(* IEC 61131-3 sources: PLC_FB_Sequencer/, 4 files *)

(* ---- MachineState1.st ---- *)
(* ======================================== *)
(* State Machine:  *)
(* Author: 1.0 *)
(* Version:  *)
(* Generated: 2025-11-28 15:15:25 *)
(* ======================================== *)

FUNCTION_BLOCK

VAR_INPUT
    IN_01 : BOOL;
    IN_02 : BOOL;
    IN_03 : BOOL;
    IN_04 : BOOL;
    IN_05 : BOOL;
    IN_06 : BOOL;
    IN_07 : BOOL;
    IN_08 : BOOL;
    IN_09 : BOOL;
    IN_10 : BOOL;
    IN_11 : BOOL;
    IN_12 : BOOL;
    IN_13 : BOOL;
    IN_14 : BOOL;
    IN_15 : BOOL;
    IN_16 : BOOL;
END_VAR

VAR_OUTPUT
    OUT_01 : BOOL;
    OUT_02 : BOOL;
    OUT_03 : BOOL;
    OUT_04 : BOOL;
    OUT_05 : BOOL;
    OUT_06 : BOOL;
    OUT_07 : BOOL;
    OUT_08 : BOOL;
    OUT_09 : BOOL;
    OUT_10 : BOOL;
    OUT_11 : BOOL;
    OUT_12 : BOOL;
    OUT_13 : BOOL;
    OUT_14 : BOOL;
    OUT_15 : BOOL;
    OUT_16 : BOOL;
END_VAR

VAR
    currentState : (IDLE, STATE_2, STATE_3) := IDLE;
END_VAR

(* State Machine Logic *)
CASE currentState OF

    IDLE:
        (* Actions *)
        OUT_01 := FALSE;
        OUT_02 := FALSE;
        OUT_03 := FALSE;
        OUT_04 := FALSE;
        OUT_05 := FALSE;
        OUT_06 := FALSE;
        OUT_07 := FALSE;
        OUT_08 := FALSE;
        OUT_09 := FALSE;
        OUT_10 := FALSE;
        OUT_11 := FALSE;
        OUT_12 := FALSE;
        OUT_13 := FALSE;
        OUT_14 := FALSE;
        OUT_15 := FALSE;
        OUT_16 := FALSE;
        (* No actions *)

        (* Transitions *)
        IF IN_01 AND IN_02 THEN  (* Example transition *)
            currentState := STATE_2;
        END_IF;

    STATE_2:
        (* Actions *)
        OUT_01 := TRUE;
        OUT_02 := FALSE;
        OUT_03 := FALSE;
        OUT_04 := FALSE;
        OUT_05 := FALSE;
        OUT_06 := FALSE;
        OUT_07 := FALSE;
        OUT_08 := FALSE;
        OUT_09 := FALSE;
        OUT_10 := FALSE;
        OUT_11 := FALSE;
        OUT_12 := FALSE;
        OUT_13 := FALSE;
        OUT_14 := FALSE;
        OUT_15 := FALSE;
        OUT_16 := FALSE;
        (* No actions *)

        (* Transitions *)
        IF IN_03 THEN
            currentState := STATE_3;
        END_IF;

    STATE_3:
        (* Actions *)
        OUT_01 := TRUE;
        OUT_02 := TRUE;
        OUT_03 := FALSE;
        OUT_04 := FALSE;
        OUT_05 := FALSE;
        OUT_06 := FALSE;
        OUT_07 := FALSE;
        OUT_08 := FALSE;
        OUT_09 := FALSE;
        OUT_10 := FALSE;
        OUT_11 := FALSE;
        OUT_12 := FALSE;
        OUT_13 := FALSE;
        OUT_14 := FALSE;
        OUT_15 := FALSE;
        OUT_16 := FALSE;
        (* No actions *)

        (* Transitions *)
        IF NOT IN_01 THEN
            currentState := IDLE;
        END_IF;
END_CASE;

END_FUNCTION_BLOCK

(* ---- MachineState2.st ---- *)
(* ======================================== *)
(* State Machine:  *)
(* Author: 1.0 *)
(* Version:  *)
(* Generated: 2025-11-29 16:41:58 *)
(* ======================================== *)

FUNCTION_BLOCK

VAR_INPUT
    IN_01 : BOOL;
    IN_02 : BOOL;
    IN_03 : BOOL;
    IN_04 : BOOL;
    IN_05 : BOOL;
    IN_06 : BOOL;
    IN_07 : BOOL;
    IN_08 : BOOL;
    IN_09 : BOOL;
    IN_10 : BOOL;
    IN_11 : BOOL;
    IN_12 : BOOL;
    IN_13 : BOOL;
    IN_14 : BOOL;
    IN_15 : BOOL;
    IN_16 : BOOL;
END_VAR

VAR_OUTPUT
    OUT_01 : BOOL;
    OUT_02 : BOOL;
    OUT_03 : BOOL;
    OUT_04 : BOOL;
    OUT_05 : BOOL;
    OUT_06 : BOOL;
    OUT_07 : BOOL;
    OUT_08 : BOOL;
    OUT_09 : BOOL;
    OUT_10 : BOOL;
    OUT_11 : BOOL;
    OUT_12 : BOOL;
    OUT_13 : BOOL;
    OUT_14 : BOOL;
    OUT_15 : BOOL;
    OUT_16 : BOOL;
END_VAR

VAR
    currentState : (IDLE, STATE_2, STATE_3) := IDLE;
END_VAR

(* State Machine Logic *)
CASE currentState OF

    IDLE:
        (* Actions *)
        OUT_01 := FALSE;
        OUT_02 := FALSE;
        OUT_03 := FALSE;
        OUT_04 := FALSE;
        OUT_05 := FALSE;
        OUT_06 := FALSE;
        OUT_07 := FALSE;
        OUT_08 := FALSE;
        OUT_09 := FALSE;
        OUT_10 := FALSE;
        OUT_11 := FALSE;
        OUT_12 := FALSE;
        OUT_13 := FALSE;
        OUT_14 := FALSE;
        OUT_15 := FALSE;
        OUT_16 := FALSE;
        (* No actions *)

        (* Transitions *)
        IF IN_01 AND IN_02 THEN  (* Example transition *)
            currentState := STATE_2;
        END_IF;

    STATE_2:
        (* Actions *)
        OUT_01 := TRUE;
        OUT_02 := FALSE;
        OUT_03 := FALSE;
        OUT_04 := FALSE;
        OUT_05 := FALSE;
        OUT_06 := FALSE;
        OUT_07 := FALSE;
        OUT_08 := FALSE;
        OUT_09 := FALSE;
        OUT_10 := FALSE;
        OUT_11 := FALSE;
        OUT_12 := FALSE;
        OUT_13 := FALSE;
        OUT_14 := FALSE;
        OUT_15 := FALSE;
        OUT_16 := FALSE;
        (* No actions *)

        (* Transitions *)
        IF IN_03 THEN
            currentState := STATE_3;
        END_IF;

    STATE_3:
        (* Actions *)
        OUT_01 := TRUE;
        OUT_02 := TRUE;
        OUT_03 := FALSE;
        OUT_04 := FALSE;
        OUT_05 := FALSE;
        OUT_06 := FALSE;
        OUT_07 := FALSE;
        OUT_08 := FALSE;
        OUT_09 := FALSE;
        OUT_10 := FALSE;
        OUT_11 := FALSE;
        OUT_12 := FALSE;
        OUT_13 := FALSE;
        OUT_14 := FALSE;
        OUT_15 := FALSE;
        OUT_16 := FALSE;
        (* No actions *)

        (* Transitions *)
        IF NOT IN_01 THEN
            currentState := IDLE;
        END_IF;
END_CASE;

END_FUNCTION_BLOCK

(* ---- MachineState3.st ---- *)
(* ======================================== *)
(* State Machine: FBSeq *)
(* Author: Gregory Brooks *)
(* Version: 1.0 *)
(* Generated: 2025-11-29 17:00:29 *)
(* ======================================== *)

FUNCTION_BLOCK FBSeq

VAR_INPUT
    IN_01 : BOOL;
    IN_02 : BOOL;
    IN_03 : BOOL;
    IN_04 : BOOL;
    IN_05 : BOOL;
    IN_06 : BOOL;
    IN_07 : BOOL;
    IN_08 : BOOL;
    IN_09 : BOOL;
    IN_10 : BOOL;
    IN_11 : BOOL;
    IN_12 : BOOL;
    IN_13 : BOOL;
    IN_14 : BOOL;
    IN_15 : BOOL;
    IN_16 : BOOL;
END_VAR

VAR_OUTPUT
    OUT_01 : BOOL;
    OUT_02 : BOOL;
    OUT_03 : BOOL;
    OUT_04 : BOOL;
    OUT_05 : BOOL;
    OUT_06 : BOOL;
    OUT_07 : BOOL;
    OUT_08 : BOOL;
    OUT_09 : BOOL;
    OUT_10 : BOOL;
    OUT_11 : BOOL;
    OUT_12 : BOOL;
    OUT_13 : BOOL;
    OUT_14 : BOOL;
    OUT_15 : BOOL;
    OUT_16 : BOOL;
END_VAR

VAR
    currentState : (IDLE, STATE_2, STATE_3) := IDLE;
END_VAR

(* State Machine Logic *)
CASE currentState OF

    IDLE:
        (* Actions *)
        OUT_01 := FALSE;
        OUT_02 := FALSE;
        OUT_03 := FALSE;
        OUT_04 := FALSE;
        OUT_05 := FALSE;
        OUT_06 := FALSE;
        OUT_07 := FALSE;
        OUT_08 := FALSE;
        OUT_09 := FALSE;
        OUT_10 := FALSE;
        OUT_11 := FALSE;
        OUT_12 := FALSE;
        OUT_13 := FALSE;
        OUT_14 := FALSE;
        OUT_15 := FALSE;
        OUT_16 := FALSE;

        (* Transitions *)
        IF IN_01 AND IN_02 THEN  (* Example transition *)
            currentState := STATE_2;
        END_IF;

    STATE_2:
        (* Actions *)
        OUT_01 := TRUE;
        OUT_02 := FALSE;
        OUT_03 := FALSE;
        OUT_04 := FALSE;
        OUT_05 := FALSE;
        OUT_06 := FALSE;
        OUT_07 := FALSE;
        OUT_08 := FALSE;
        OUT_09 := FALSE;
        OUT_10 := FALSE;
        OUT_11 := FALSE;
        OUT_12 := FALSE;
        OUT_13 := FALSE;
        OUT_14 := FALSE;
        OUT_15 := FALSE;
        OUT_16 := FALSE;

        (* Transitions *)
        IF IN_03 THEN
            currentState := STATE_3;
        END_IF;

    STATE_3:
        (* Actions *)
        OUT_01 := TRUE;
        OUT_02 := TRUE;
        OUT_03 := FALSE;
        OUT_04 := FALSE;
        OUT_05 := FALSE;
        OUT_06 := FALSE;
        OUT_07 := FALSE;
        OUT_08 := FALSE;
        OUT_09 := FALSE;
        OUT_10 := FALSE;
        OUT_11 := FALSE;
        OUT_12 := FALSE;
        OUT_13 := FALSE;
        OUT_14 := FALSE;
        OUT_15 := FALSE;
        OUT_16 := FALSE;

        (* Transitions *)
        IF NOT IN_01 THEN
            currentState := IDLE;
        END_IF;
END_CASE;

END_FUNCTION_BLOCK

(* ---- PRG_CrimpDevice.st ---- *)
(* ======================================== *)
(* Wrapper program for FB_CrimpDeviceSeq *)
(* Runs the timers externally and maps physical I/O. *)
(* FB_CrimpDeviceSeq is generated from CrimpDevice_StateMachine.fods *)
(* ======================================== *)

PROGRAM PRG_CrimpDevice

VAR
    S1Start AT %IX0.0 : BOOL;   (* Start button *)
    S2Confirm AT %IX0.1 : BOOL; (* Unload confirmation button *)
    qxA1Crimp AT %QX0.0 : BOOL; (* Crimp actuator *)
    qxP1Unload AT %QX0.1 : BOOL; (* Unload actuator *)

    G_CrimpDevice : FB_CrimpDeviceSeq;
    tX2 : TON;  (* Crimp time *)
    tX3 : TON;  (* Pause time *)
END_VAR

(* Timers are driven by the step flag outputs of the state machine *)
tX2(IN := G_CrimpDevice.X2, PT := T#2S);
tX3(IN := G_CrimpDevice.X3, PT := T#5S);

G_CrimpDevice(
    S1Start := S1Start,
    S2Confirm := S2Confirm,
    T1CrimpDone := tX2.Q,
    T2PauseDone := tX3.Q);

(* Refresh the physical output image *)
qxA1Crimp := G_CrimpDevice.A1Crimp;
qxP1Unload := G_CrimpDevice.P1Unload;

END_PROGRAM
